ACTION A_Home:
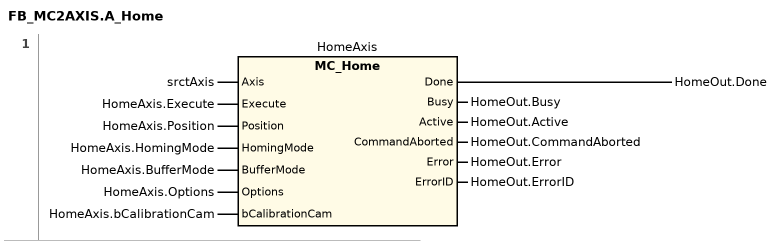
// NETWORK 1
HomeAxis(
    Axis := srctAxis,
    Execute := HomeAxis.Execute,
    Position := HomeAxis.Position,
    HomingMode := HomeAxis.HomingMode,
    BufferMode := HomeAxis.BufferMode,
    Options := HomeAxis.Options,
    bCalibrationCam := HomeAxis.bCalibrationCam,
    Busy => HomeOut.Busy,
    Active => HomeOut.Active,
    CommandAborted => HomeOut.CommandAborted,
    Error => HomeOut.Error,
    ErrorID => HomeOut.ErrorID); // MC_Home
HomeOut.Done := HomeAxis.Done;
END_ACTION

ACTION A_Jog:
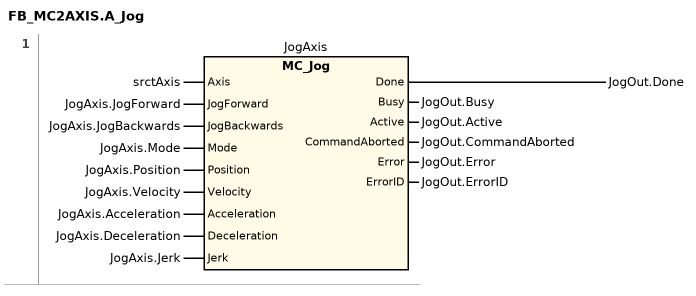
// NETWORK 1
JogAxis(
    Axis := srctAxis,
    JogForward := JogAxis.JogForward,
    JogBackwards := JogAxis.JogBackwards,
    Mode := JogAxis.Mode,
    Position := JogAxis.Position,
    Velocity := JogAxis.Velocity,
    Acceleration := JogAxis.Acceleration,
    Deceleration := JogAxis.Deceleration,
    Jerk := JogAxis.Jerk,
    Busy => JogOut.Busy,
    Active => JogOut.Active,
    CommandAborted => JogOut.CommandAborted,
    Error => JogOut.Error,
    ErrorID => JogOut.ErrorID); // MC_Jog
JogOut.Done := JogAxis.Done;
END_ACTION

ACTION A_MovAbs:
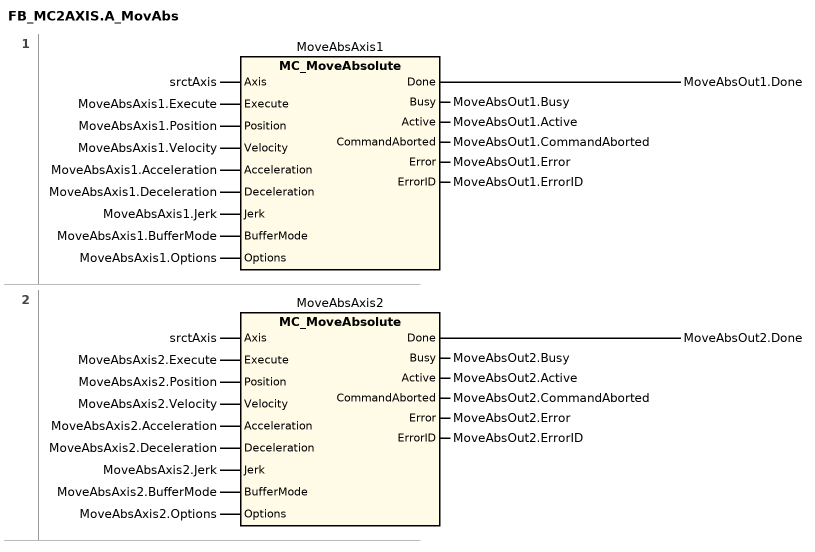
// NETWORK 1
MoveAbsAxis1(
    Axis := srctAxis,
    Execute := MoveAbsAxis1.Execute,
    Position := MoveAbsAxis1.Position,
    Velocity := MoveAbsAxis1.Velocity,
    Acceleration := MoveAbsAxis1.Acceleration,
    Deceleration := MoveAbsAxis1.Deceleration,
    Jerk := MoveAbsAxis1.Jerk,
    BufferMode := MoveAbsAxis1.BufferMode,
    Options := MoveAbsAxis1.Options,
    Busy => MoveAbsOut1.Busy,
    Active => MoveAbsOut1.Active,
    CommandAborted => MoveAbsOut1.CommandAborted,
    Error => MoveAbsOut1.Error,
    ErrorID => MoveAbsOut1.ErrorID); // MC_MoveAbsolute
MoveAbsOut1.Done := MoveAbsAxis1.Done;

// NETWORK 2
MoveAbsAxis2(
    Axis := srctAxis,
    Execute := MoveAbsAxis2.Execute,
    Position := MoveAbsAxis2.Position,
    Velocity := MoveAbsAxis2.Velocity,
    Acceleration := MoveAbsAxis2.Acceleration,
    Deceleration := MoveAbsAxis2.Deceleration,
    Jerk := MoveAbsAxis2.Jerk,
    BufferMode := MoveAbsAxis2.BufferMode,
    Options := MoveAbsAxis2.Options,
    Busy => MoveAbsOut2.Busy,
    Active => MoveAbsOut2.Active,
    CommandAborted => MoveAbsOut2.CommandAborted,
    Error => MoveAbsOut2.Error,
    ErrorID => MoveAbsOut2.ErrorID); // MC_MoveAbsolute
MoveAbsOut2.Done := MoveAbsAxis2.Done;
END_ACTION

ACTION A_MovAdd:
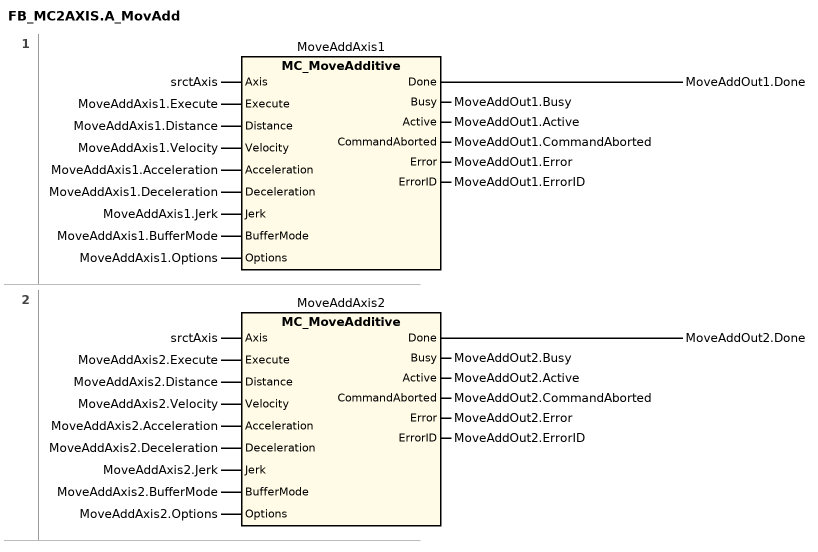
// NETWORK 1
MoveAddAxis1(
    Axis := srctAxis,
    Execute := MoveAddAxis1.Execute,
    Distance := MoveAddAxis1.Distance,
    Velocity := MoveAddAxis1.Velocity,
    Acceleration := MoveAddAxis1.Acceleration,
    Deceleration := MoveAddAxis1.Deceleration,
    Jerk := MoveAddAxis1.Jerk,
    BufferMode := MoveAddAxis1.BufferMode,
    Options := MoveAddAxis1.Options,
    Busy => MoveAddOut1.Busy,
    Active => MoveAddOut1.Active,
    CommandAborted => MoveAddOut1.CommandAborted,
    Error => MoveAddOut1.Error,
    ErrorID => MoveAddOut1.ErrorID); // MC_MoveAdditive
MoveAddOut1.Done := MoveAddAxis1.Done;

// NETWORK 2
MoveAddAxis2(
    Axis := srctAxis,
    Execute := MoveAddAxis2.Execute,
    Distance := MoveAddAxis2.Distance,
    Velocity := MoveAddAxis2.Velocity,
    Acceleration := MoveAddAxis2.Acceleration,
    Deceleration := MoveAddAxis2.Deceleration,
    Jerk := MoveAddAxis2.Jerk,
    BufferMode := MoveAddAxis2.BufferMode,
    Options := MoveAddAxis2.Options,
    Busy => MoveAddOut2.Busy,
    Active => MoveAddOut2.Active,
    CommandAborted => MoveAddOut2.CommandAborted,
    Error => MoveAddOut2.Error,
    ErrorID => MoveAddOut2.ErrorID); // MC_MoveAdditive
MoveAddOut2.Done := MoveAddAxis2.Done;
END_ACTION

ACTION A_MovMod:
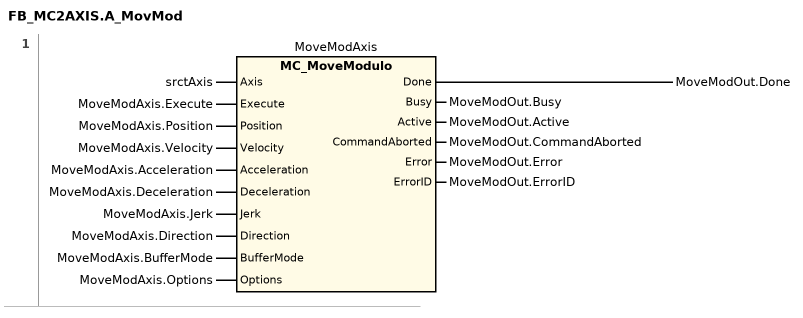
// NETWORK 1
MoveModAxis(
    Axis := srctAxis,
    Execute := MoveModAxis.Execute,
    Position := MoveModAxis.Position,
    Velocity := MoveModAxis.Velocity,
    Acceleration := MoveModAxis.Acceleration,
    Deceleration := MoveModAxis.Deceleration,
    Jerk := MoveModAxis.Jerk,
    Direction := MoveModAxis.Direction,
    BufferMode := MoveModAxis.BufferMode,
    Options := MoveModAxis.Options,
    Busy => MoveModOut.Busy,
    Active => MoveModOut.Active,
    CommandAborted => MoveModOut.CommandAborted,
    Error => MoveModOut.Error,
    ErrorID => MoveModOut.ErrorID); // MC_MoveModulo
MoveModOut.Done := MoveModAxis.Done;
END_ACTION

ACTION A_MovRel:
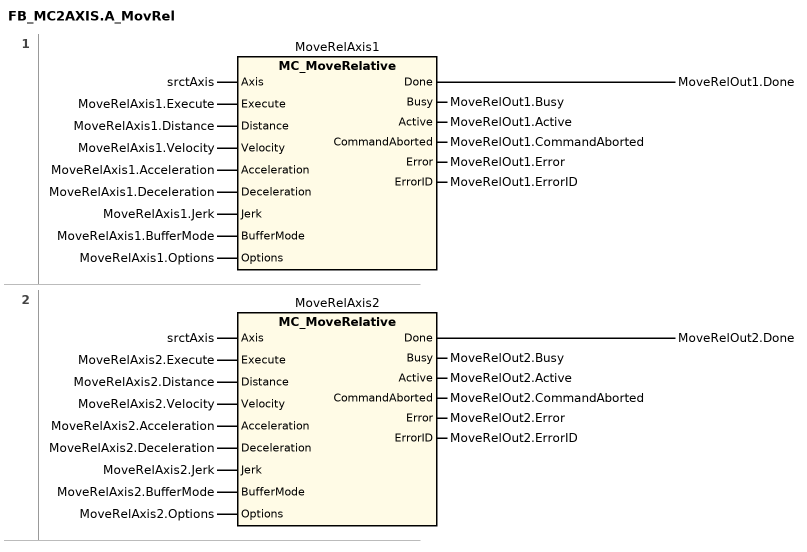
// NETWORK 1
MoveRelAxis1(
    Axis := srctAxis,
    Execute := MoveRelAxis1.Execute,
    Distance := MoveRelAxis1.Distance,
    Velocity := MoveRelAxis1.Velocity,
    Acceleration := MoveRelAxis1.Acceleration,
    Deceleration := MoveRelAxis1.Deceleration,
    Jerk := MoveRelAxis1.Jerk,
    BufferMode := MoveRelAxis1.BufferMode,
    Options := MoveRelAxis1.Options,
    Busy => MoveRelOut1.Busy,
    Active => MoveRelOut1.Active,
    CommandAborted => MoveRelOut1.CommandAborted,
    Error => MoveRelOut1.Error,
    ErrorID => MoveRelOut1.ErrorID); // MC_MoveRelative
MoveRelOut1.Done := MoveRelAxis1.Done;

// NETWORK 2
MoveRelAxis2(
    Axis := srctAxis,
    Execute := MoveRelAxis2.Execute,
    Distance := MoveRelAxis2.Distance,
    Velocity := MoveRelAxis2.Velocity,
    Acceleration := MoveRelAxis2.Acceleration,
    Deceleration := MoveRelAxis2.Deceleration,
    Jerk := MoveRelAxis2.Jerk,
    BufferMode := MoveRelAxis2.BufferMode,
    Options := MoveRelAxis2.Options,
    Busy => MoveRelOut2.Busy,
    Active => MoveRelOut2.Active,
    CommandAborted => MoveRelOut2.CommandAborted,
    Error => MoveRelOut2.Error,
    ErrorID => MoveRelOut2.ErrorID); // MC_MoveRelative
MoveRelOut2.Done := MoveRelAxis2.Done;
END_ACTION

ACTION A_MovVel:
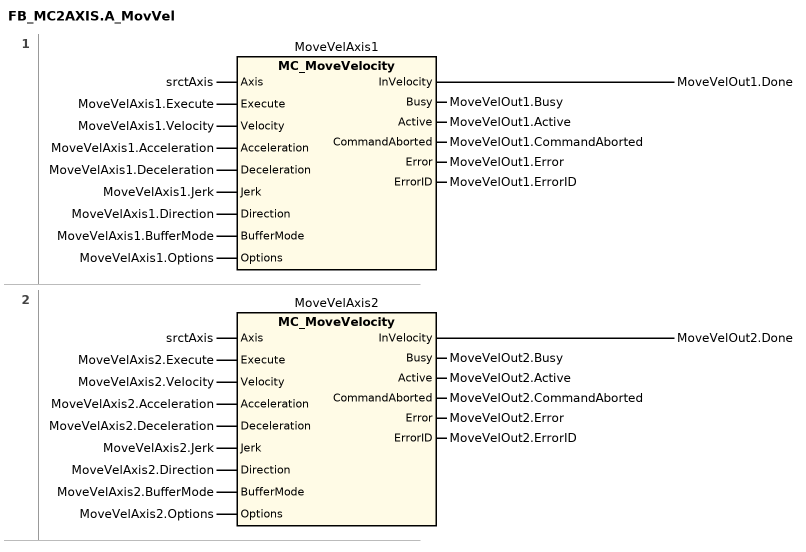
// NETWORK 1
MoveVelAxis1(
    Axis := srctAxis,
    Execute := MoveVelAxis1.Execute,
    Velocity := MoveVelAxis1.Velocity,
    Acceleration := MoveVelAxis1.Acceleration,
    Deceleration := MoveVelAxis1.Deceleration,
    Jerk := MoveVelAxis1.Jerk,
    Direction := MoveVelAxis1.Direction,
    BufferMode := MoveVelAxis1.BufferMode,
    Options := MoveVelAxis1.Options,
    Busy => MoveVelOut1.Busy,
    Active => MoveVelOut1.Active,
    CommandAborted => MoveVelOut1.CommandAborted,
    Error => MoveVelOut1.Error,
    ErrorID => MoveVelOut1.ErrorID); // MC_MoveVelocity
MoveVelOut1.Done := MoveVelAxis1.InVelocity;

// NETWORK 2
MoveVelAxis2(
    Axis := srctAxis,
    Execute := MoveVelAxis2.Execute,
    Velocity := MoveVelAxis2.Velocity,
    Acceleration := MoveVelAxis2.Acceleration,
    Deceleration := MoveVelAxis2.Deceleration,
    Jerk := MoveVelAxis2.Jerk,
    Direction := MoveVelAxis2.Direction,
    BufferMode := MoveVelAxis2.BufferMode,
    Options := MoveVelAxis2.Options,
    Busy => MoveVelOut2.Busy,
    Active => MoveVelOut2.Active,
    CommandAborted => MoveVelOut2.CommandAborted,
    Error => MoveVelOut2.Error,
    ErrorID => MoveVelOut2.ErrorID); // MC_MoveVelocity
MoveVelOut2.Done := MoveVelAxis2.InVelocity;
END_ACTION

ACTION A_Power:

(* read in parameters from the AX5000 via SoE, Reset via SoE *)
fbPowerAxis(
	Enable			:= bEnableAxis,
	Enable_Positive	:= bEnablePos,
	Enable_Negative	:= bEnableNeg,
	Override		:= fOverride,
	Axis			:= srctAxis,
	);

PowerAxisOut.Done := fbPowerAxis.Status;
PowerAxisOut.Busy := fbPowerAxis.Busy;
PowerAxisOut.Active := fbPowerAxis.Active;
PowerAxisOut.Error := fbPowerAxis.Error;
PowerAxisOut.ErrorID := fbPowerAxis.ErrorID;
END_ACTION

ACTION A_ResMovExecute:
HomeAxis.Execute := FALSE;
MoveAbsAxis1.Execute := FALSE;
MoveAbsAxis2.Execute := FALSE;
MoveRelAxis1.Execute := FALSE;
MoveRelAxis2.Execute := FALSE;
MoveAddAxis1.Execute :=FALSE;
MoveAddAxis2.Execute :=FALSE;
MoveVelAxis1.Execute := FALSE;
MoveVelAxis2.Execute := FALSE;
MoveModAxis.Execute := FALSE;
JogAxis.JogBackwards := FALSE;
JogAxis.JogForward := FALSE;
bJogBackwards := FALSE;
bJogForward := FALSE;
END_ACTION

ACTION A_SetPosition:
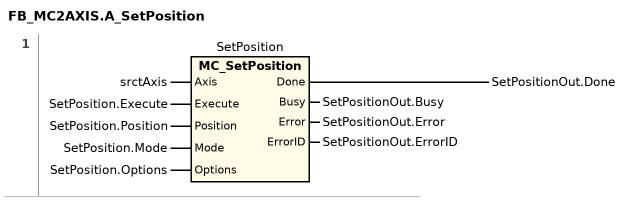
// NETWORK 1
SetPosition(
    Axis := srctAxis,
    Execute := SetPosition.Execute,
    Position := SetPosition.Position,
    Mode := SetPosition.Mode,
    Options := SetPosition.Options,
    Busy => SetPositionOut.Busy,
    Error => SetPositionOut.Error,
    ErrorID => SetPositionOut.ErrorID); // MC_SetPosition
SetPositionOut.Done := SetPosition.Done;
END_ACTION

ACTION A_Stop:
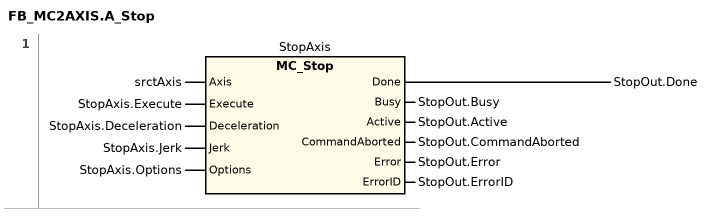
// NETWORK 1
StopAxis(
    Axis := srctAxis,
    Execute := StopAxis.Execute,
    Deceleration := StopAxis.Deceleration,
    Jerk := StopAxis.Jerk,
    Options := StopAxis.Options,
    Busy => StopOut.Busy,
    Active => StopOut.Active,
    CommandAborted => StopOut.CommandAborted,
    Error => StopOut.Error,
    ErrorID => StopOut.ErrorID); // MC_Stop
StopOut.Done := StopAxis.Done;
END_ACTION

ACTION A_Tourque:
(* Tourque and floating axis *)

FromMc2.fActMoment := IiCurrentTourque / 10;

QiTourqueMax := ABS(REAL_TO_INT(fMaxMom * 10));

IF NOT bError AND NOT FromMc2.bError AND srctAxis.Status.Operational AND FloatingCmd.bFloatingOn THEN
	(*	only floating without movement	*)
	IF NOT FloatingCmd.bPush THEN
		fbFloatingAbsAxis1(Execute := FALSE , Axis:=srctAxis);
		fbFloatingAbsAxis2(Execute := FALSE , Axis:=srctAxis);
		fbResetAxisFloating(Execute := (enState = Mc2AxisStateIdle)   , Axis := srctAxis);	(*	AND NOT srctAxis.Status.HasJob	*)
		tonResetFloating(IN := fbResetAxisFloating.Done , PT := T#30ms);
		IF tonResetFloating.Q THEN
			tonResetFloating(IN := FALSE);
			fbResetAxisFloating(Execute := FALSE, Axis := srctAxis);
		END_IF

	(*	floating with negative movement (push)	*)
	ELSIF FloatingCmd.bPush THEN
		fbFloatingMoveTrig(IN := (enState = Mc2AxisStateIdle) , PT := T#200ms);
		IF fbFloatingMoveTrig.Qr THEN
			fbFloatingMoveTrig(IN := FALSE);
			(* FB1 bevorzugen *)
			(* Busy ist high, wenn ein Befehl ansteht; Active ist high, wenn der Mov-Befehl ausgeführt wird *)
			IF NOT fbFloatingAbsAxis1.Busy THEN
				fbFloatingAbsAxis1.Position := srctAxis.NcToPlc.ActPos + FloatingCmd.fPushPos;
				fbFloatingAbsAxis1.Velocity := FloatingCmd.fPushVel;
				fbFloatingAbsAxis1(Execute := TRUE , Axis:=srctAxis);
				fbFloatingAbsAxis2(Execute := FALSE , Axis:=srctAxis);
			(* wenn FB1 aktiv -> neues Kommando mit FB2 überlagern *)
			ELSIF NOT fbFloatingAbsAxis2.Busy THEN
				fbFloatingAbsAxis2.Position := srctAxis.NcToPlc.ActPos + FloatingCmd.fPushPos;
				fbFloatingAbsAxis2.Velocity := FloatingCmd.fPushVel;
				fbFloatingAbsAxis2(Execute := TRUE , Axis:=srctAxis);
				fbFloatingAbsAxis1(Execute := FALSE , Axis:=srctAxis);
			END_IF;
			IF fbFloatingAbsAxis1.Done OR fbFloatingAbsAxis1.CommandAborted OR fbFloatingAbsAxis1.Error THEN
				fbFloatingAbsAxis1(Execute := FALSE , Axis:=srctAxis);
			END_IF
			IF fbFloatingAbsAxis2.Done OR fbFloatingAbsAxis2.CommandAborted OR fbFloatingAbsAxis2.Error THEN
				fbFloatingAbsAxis2(Execute := FALSE , Axis:=srctAxis);
			END_IF
		END_IF
	ELSE
		fbFloatingMoveTrig(IN := FALSE);
		fbFloatingAbsAxis1(Execute := FALSE , Axis:=srctAxis);
		fbFloatingAbsAxis2(Execute := FALSE , Axis:=srctAxis);
	END_IF

	bFederOffReset := FALSE;
ELSE
	fbFloatingMoveTrig(IN := FALSE);
	fbFloatingAbsAxis1(Execute := FALSE , Axis:=srctAxis);
	fbFloatingAbsAxis2(Execute := FALSE , Axis:=srctAxis);
	tonResetFloating(IN := FALSE);
	fbResetAxisFloating(Execute := FALSE, Axis := srctAxis);
	IF NOT bFederOffReset THEN
		fbResetAxisFloating(Execute := TRUE, Axis := srctAxis);
	END_IF
	bFederOffReset := TRUE;
END_IF
fbFloatingAbsAxis1(Axis:=srctAxis );
fbFloatingAbsAxis2(Axis:=srctAxis );
END_ACTION

END_FUNCTION_BLOCK

// Utilities/FB_TON_RMTH
///
///	Dieser Baustein verzögert ein Signal und gibt positive und negative Flanke dieses Signals aus
///	von Roland Ertl / www.rmth.at / 2009
FUNCTION_BLOCK FB_TON_RMTH
VAR_INPUT
	///	Signal	
	IN: BOOL;
	///	Verzögerungszeit	
	PT: TIME := TIME#100ms;
END_VAR
VAR_OUTPUT
	///	Verzögertes Signal	
	Q: BOOL;
	///	Flanken -> nur für 1 Zyklus aktiv	
	Qr: BOOL;
	///	Flanken -> nur für 1 Zyklus aktiv	
	Qf: BOOL;
END_VAR
VAR
	ton_On: TON;
	rtrig_Pos: R_TRIG;
	ftrig_Neg: F_TRIG;
END_VAR

ton_On(IN:= IN , PT:= PT , Q=> Q , ET=> );
rtrig_Pos(CLK:= ton_On.Q , Q=> Qr );
ftrig_Neg(CLK:= ton_On.Q , Q=> Qf);

END_FUNCTION_BLOCK

// Utilities/Balluff/F_GetBalluffWegValue
FUNCTION F_GetBalluffWegValue : REAL
VAR_INPUT
	/// Eingangsdaten von Wegaufnehmer
	arrBytesWeg		:ARRAY[0..3] OF BYTE;
END_VAR
VAR
	nWegTemp		:DWORD;
END_VAR

(*
	Funktion zum mappen der Speicherdaten eines Balluff Wegaufnehmers
	von www.rmth.at/ Roland Ertl / 2015
	Aufloesung 1/1000
	
**********************************************************************)

nWegTemp.0 := arrBytesWeg[3].0;
nWegTemp.1 := arrBytesWeg[3].1;
nWegTemp.2 := arrBytesWeg[3].2;
nWegTemp.3 := arrBytesWeg[3].3;
nWegTemp.4 := arrBytesWeg[3].4;
nWegTemp.5 := arrBytesWeg[3].5;
nWegTemp.6 := arrBytesWeg[3].6;
nWegTemp.7 := arrBytesWeg[3].7;

nWegTemp.8 := arrBytesWeg[2].0;
nWegTemp.9 := arrBytesWeg[2].1;
nWegTemp.10 := arrBytesWeg[2].2;
nWegTemp.11 := arrBytesWeg[2].3;
nWegTemp.12 := arrBytesWeg[2].4;
nWegTemp.13 := arrBytesWeg[2].5;
nWegTemp.14 := arrBytesWeg[2].6;
nWegTemp.15 := arrBytesWeg[2].7;


nWegTemp.16 := arrBytesWeg[1].0;
nWegTemp.17 := arrBytesWeg[1].1;
nWegTemp.18 := arrBytesWeg[1].2;
nWegTemp.19 := arrBytesWeg[1].3;
nWegTemp.20 := arrBytesWeg[1].4;
nWegTemp.21 := arrBytesWeg[1].5;
nWegTemp.22 := arrBytesWeg[1].6;
nWegTemp.23 := arrBytesWeg[1].7;

nWegTemp.24 := arrBytesWeg[0].0;
nWegTemp.25 := arrBytesWeg[0].1;
nWegTemp.26 := arrBytesWeg[0].2;
nWegTemp.27 := arrBytesWeg[0].3;
nWegTemp.28 := arrBytesWeg[0].4;
nWegTemp.29 := arrBytesWeg[0].5;
nWegTemp.30 := arrBytesWeg[0].6;
nWegTemp.31 := arrBytesWeg[0].7;


F_GetBalluffWegValue := DWORD_TO_REAL(nWegTemp) / 1000;

END_FUNCTION

// Utilities/Log/Base/FB_LoggingProviderBase
FUNCTION_BLOCK FB_LoggingProviderBase IMPLEMENTS ITFLoggingProvider

/// Add log method
{attribute '' := ''}
{attribute 'object_name' := 'AddLog'}
METHOD AddLog : BOOL
VAR_INPUT
	/// log message 
	{attribute '' := ''}
	sText: Tc2_System.T_MaxString;
	/// log source
	{attribute '' := ''}
	sSource: STRING;
	///	level: eLogLevelNone, eLogLevelError, eLogLevelWarning, eLogLevelInformation	
	{attribute '' := ''}
	eLevel: E_LogLevel;
END_VAR
VAR
	idx: INT;
END_VAR
///
/// Funktionen zum Hinzufuegen einer Log-Nachricht
/// Rueckgabe: TRUE, bei Erfolg, anderenfalls FALSE
/// 17.05.2010		www.rmth.at
///

idx := iLogArraySize;
REPEAT
	arLoggs[idx] := arLoggs[idx - 1];
    idx:= idx - 1;
UNTIL
    	idx = 0
END_REPEAT

arLoggs[0].sText:= sText;
arLoggs[0].sSource:= sSource;
arLoggs[0].bSaveRequest := TRUE;
arLoggs[0].bSaved  := FALSE;
arLoggs[0].eLevel := eLevel;
arLoggs[0].sTime := sTimeString;

//	Return Result
AddLog := TRUE;
END_METHOD

{attribute 'object_name' := 'Run'}
METHOD Run
END_METHOD

END_FUNCTION_BLOCK

// Utilities/Log/Interface/ITFLoggingProvider
INTERFACE ITFLoggingProvider

/// Add log method
{attribute 'object_name' := 'AddLog'}
METHOD AddLog : BOOL
VAR_INPUT
	/// log message 
	sText: T_MaxString;
	/// log source
	sSource: STRING;
	///	level: eLogLevelNone, eLogLevelError, eLogLevelWarning, eLogLevelInformation	
	eLevel: E_LogLevel;
END_VAR
END_METHOD

{attribute 'object_name' := 'Run'}
METHOD Run
END_METHOD

END_INTERFACE

// Utilities/Log/FB_DebugLoggingProvider
///Funktionblock zum Loggen
FUNCTION_BLOCK FB_DebugLoggingProvider EXTENDS FB_LoggingProviderBase
VAR_IN_OUT
	stLogConfig: ST_LoggingConfig;
END_VAR

///
/// Funktionblock zum Loggen - nur in array
/// 17.05.2010 www.rmth.at
///

END_FUNCTION_BLOCK

// Utilities/Log/FB_EventLoggingProvider
///Funktionblock zum Loggen
FUNCTION_BLOCK FB_EventLoggingProvider EXTENDS FB_LoggingProviderBase
VAR_IN_OUT
	stLogConfig: ST_LoggingConfig;
END_VAR
VAR
	///	logg Message	
	bLoggMessage: BOOL;
	///	input structure		
	strctLogging: ST_Log;
	toiLogging: TON;
	timeLogging: TIME := TIME#2s0ms;
	iLogging: INT;
	ii: INT;
	iSave: INT;
	stEmpty: ST_Log;
	///	MESSAGE ON				
	rtrig_IN: R_TRIG;
	///	message type				
	msgCtrlMask: DWORD;
	///	logging text					
	sText: T_MaxString;
END_VAR

///
/// Funktionblock zum Loggen - windows event log
/// 17.05.2010 www.rmth.at
///

ACTION EventLog:

(*	log trigger	*)
rtrig_IN(clk:= bLoggMessage);

(*	no Log from Configuration	*)
IF stLogConfig.eLogLevel = eLogLevelNone THEN
	bLoggMessage := FALSE;
	RETURN;
END_IF

// switch level
CASE stLogConfig.eLogLevel OF
	eLogLevelInformation:	(*	all eKinds	*)
		IF strctLogging.eLevel = eLogLevelNone THEN
			bLoggMessage := FALSE;
			RETURN;
		END_IF
		
	eLogLevelWarning: 		(*	only Error and Warning	*)
		IF strctLogging.eLevel = eLogLevelNone OR strctLogging.eLevel = eLogLevelInformation THEN
			bLoggMessage := FALSE;
			RETURN;
		END_IF
		
	eLogLevelError: 	(*	only Error	*)
		IF strctLogging.eLevel = eLogLevelNone OR strctLogging.eLevel = eLogLevelInformation OR strctLogging.eLevel = eLogLevelWarning THEN
			bLoggMessage := FALSE;
			RETURN;
		END_IF
		
	ELSE (*	default = none		*)
		bLoggMessage := FALSE;
		RETURN;
		
END_CASE

(*	Event Logg	*)
CASE strctLogging.eLevel OF
	eLogLevelError:	
		msgCtrlMask := 16#14 ; 	(*	Error		*)
	eLogLevelWarning:	
		msgCtrlMask := 16#12;  	(*	Warning		*)
	eLogLevelInformation:
		msgCtrlMask := 16#11;  	(*	Information	*)
ELSE
	msgCtrlMask := 16#11;  	(*	default: Information	*)
END_CASE

IF rtrig_IN.Q THEN
	sText  := strctLogging.sTime;
	sText := CONCAT( sText, ':');
	sText := CONCAT( sText, strctLogging.sSource);
	sText := CONCAT( sText, ':');
	sText := CONCAT( sText, strctLogging.sText);
	ADSLOGSTR(msgCtrlMask,   sText   , '');
END_IF
END_ACTION

ACTION Logger:
///
/// Programm for Logging Messages
/// 11.05.2012	www.rmth.at
///

toiLogging(PT:= timeLogging);

CASE iLogging OF

	0: (*	wait initial Time	*)
		toiLogging.IN := TRUE;
		IF toiLogging.Q THEN
			toiLogging.IN:= FALSE;
			iSave:= 0;
			ii:= 500;
			iLogging := iLogging + 1;
		END_IF

	1: (*	iSave all messages in array list	*)
		CASE iSave OF
			0: 	IF arLoggs[ii].bSaveRequest THEN
					IF  NOT arLoggs[ii].bSaved THEN
						iSave := 10;
					ELSE
						iSave := 100;
					END_IF
				ELSE
					iSave := 100;
				END_IF
	
			10: 	(*	iSave message	*)
				strctLogging := arLoggs[ii];
				bLoggMessage := TRUE;
				iSave:= 11;
	
			11: 	(*	check iSaved	*)
				IF NOT bLoggMessage THEN
					arLoggs[ii].bSaved := TRUE;
					arLoggs[ii].bSaveRequest := FALSE;
					iSave := 100;
				END_IF
	
			100: 	(*	decrement	*)
				ii:= ii - 1;
				iSave := 101;
	
			101:
				IF ii < 0 THEN	(*	all messages checked	*)
					iLogging := iLogging + 1;	(*	next step == clear	*)
				ELSE
					iSave:=0;
				END_IF
		END_CASE

	2: 	(*	delete all iSaved messages	*)
		FOR ii:=0 TO 500 BY 1 DO
			IF arLoggs[ii].bSaved AND NOT arLoggs[ii].bSaveRequest THEN
				arLoggs[ii] := stEmpty;
			END_IF
		END_FOR
		iLogging := 0;

END_CASE
END_ACTION

{attribute 'object_name' := 'Run'}
METHOD Run
Logger();
EventLog();
END_METHOD

END_FUNCTION_BLOCK

// Utilities/Log/FB_FileLoggingProvider
///Funktionblock zum Loggen
FUNCTION_BLOCK FB_FileLoggingProvider EXTENDS FB_LoggingProviderBase
VAR_IN_OUT
	stLogConfig: ST_LoggingConfig;
END_VAR
VAR
	iInit: INT;
	///	logg Message	
	bLoggMessage: BOOL;
	///	input structure		
	strctLogging: ST_Log;
	///	file path example c:\Daten\PLC exist	
	bFilePathExist: BOOL;
	toiLogging: TON;
	timeLogging: TIME := TIME#2s0ms;
	iLogging: INT;
	ii: INT;
	iSave: INT;
	stEmpty: ST_Log;
	///	MESSAGE ON				
	rtrig_IN: R_TRIG;
	///	logging text					
	sText: T_MaxString;
	///	step flow file logging	
	iStepFileLogging: INT;
	hFile: UINT;
	///	full path				
	sPath: STRING;
	///	new full path			
	sPathNew: STRING;
	///	fbs	
	fbFileOpen: FB_FileOpen;
	fbFileWrite: FB_FileWrite;
	bFileWriteBusy: BOOL;
	bFileWriteError: BOOL;
	nFileWriteErrorId: UDINT;
	nFileWriteCount: UDINT;
	fbFileClose: FB_FileClose;
	bFileCloseBusy: BOOL;
	bFileCloseError: BOOL;
	nFileCloseErrorId: UDINT;
	fbEOF: FB_EOF;
	bEOFBusy: BOOL;
	bEOFError: BOOL;
	nEOFErrorId: UDINT;
	///	max file size	
	bIsEOF: BOOL;
	fbFileRename: FB_FileRename;
	bFileRename: BOOL;
	bFileRenameBusy: BOOL;
	bFileRenameError: BOOL;
	nFileRenameErrId: UDINT;
END_VAR

///
/// Funktionblock zum Loggen in Datei
/// 17.05.2010 www.rmth.at
///

{attribute 'object_name' := 'Initialize'}
METHOD PRIVATE Initialize

P_FilePath();

CASE iInit OF
	0:	// path name from configuration
		P_FilePath.sPathName := stLogConfig.sLogPath;
		P_FilePath.bCreateDIR := TRUE;
		iInit := 10;
		
	10:	// wait for folder exists
		IF P_FilePath.bFolderExist THEN
			bFilePathExist := TRUE;
			P_FilePath.bCreateDIR := FALSE;
			iInit := 0;
		END_IF		
END_CASE
END_METHOD

ACTION Logger:
///
/// Programm for Logging Messages
/// 11.05.2012	www.rmth.at
///

toiLogging(PT:= timeLogging);

CASE iLogging OF

	0: (*	wait initial Time	*)
		toiLogging.IN := TRUE;
		IF toiLogging.Q THEN
			toiLogging.IN:= FALSE;
			iSave:= 0;
			ii:= 500;
			iLogging := iLogging + 1;
		END_IF

	1: (*	iSave all messages in array list	*)
		CASE iSave OF
			0: 	IF arLoggs[ii].bSaveRequest THEN
					IF  NOT arLoggs[ii].bSaved THEN
						iSave := 10;
					ELSE
						iSave := 100;
					END_IF
				ELSE
					iSave := 100;
				END_IF
	
			10: 	(*	iSave message	*)
				strctLogging := arLoggs[ii];
				bLoggMessage := TRUE;
				iSave:= 11;
	
			11: 	(*	check iSaved	*)
				IF NOT bLoggMessage THEN
					arLoggs[ii].bSaved := TRUE;
					arLoggs[ii].bSaveRequest := FALSE;
					iSave := 100;
				END_IF
	
			100: 	(*	decrement	*)
				ii:= ii - 1;
				iSave := 101;
	
			101:
				IF ii < 0 THEN	(*	all messages checked	*)
					iLogging := iLogging + 1;	(*	next step == clear	*)
				ELSE
					iSave:=0;
				END_IF
		END_CASE

	2: 	(*	delete all iSaved messages	*)
		FOR ii:=0 TO 500 BY 1 DO
			IF arLoggs[ii].bSaved AND NOT arLoggs[ii].bSaveRequest THEN
				arLoggs[ii] := stEmpty;
			END_IF
		END_FOR
		iLogging := 0;

END_CASE
END_ACTION

{attribute 'object_name' := 'Run'}
METHOD Run
IF NOT bFilePathExist THEN
	Initialize();	
	RETURN;
END_IF

Logger();
WriteFile();
END_METHOD

ACTION WriteFile:

(*	run function logging	*)

(*	trigger	*)
rtrig_IN(clk:= bLoggMessage);

(*	no Log from Configuration	*)
IF stLogConfig.eLogLevel = eLogLevelNone THEN
	bLoggMessage := FALSE;
	RETURN;
END_IF

CASE stLogConfig.eLogLevel OF
	eLogLevelInformation:	(*	all eKinds	*)
		IF strctLogging.eLevel = eLogLevelNone THEN
			bLoggMessage := FALSE;
			RETURN;
		END_IF
	eLogLevelWarning: 		(*	only Error and Warning	*)
		IF strctLogging.eLevel = eLogLevelNone OR strctLogging.eLevel = eLogLevelInformation THEN
			bLoggMessage := FALSE;
			RETURN;
		END_IF
	eLogLevelError: 	(*	only Error	*)
		IF strctLogging.eLevel = eLogLevelNone OR strctLogging.eLevel = eLogLevelInformation OR strctLogging.eLevel = eLogLevelWarning THEN
			bLoggMessage := FALSE;
			RETURN;
		END_IF
	ELSE (*	default = none		*)
		bLoggMessage := FALSE;
		RETURN;
END_CASE

(*	FILE LOG	*)
sPath := '';
sPath := CONCAT(stLogConfig.sLogPath, '\');
sPath := CONCAT(sPath, stLogConfig.sLogName);

sPathNew := '';
sPathNew := CONCAT(stLogConfig.sLogPath, '\');
(*sTimeString:= DELETE(sTimeString,10,10);*)

sPathNew := CONCAT(sPathNew, sTimeString);
sPathNew := CONCAT(sPathNew,'.log');

IF bFilePathExist THEN

	CASE strctLogging.eLevel OF
		eLogLevelError:			(*	Erro		*)
			sText := '$R$N ERR ';
		eLogLevelWarning:		(*	Warning		*)	
			sText := '$R$N WARN ';
		eLogLevelInformation:	(*	info		*)	
			sText := '$R$N INF ';
	ELSE						(*	default		*)				
			sText := '$R$N INF ';
	END_CASE

	sText := CONCAT(sText, strctLogging.sTime);
	sText := CONCAT(sText, ' ');
	sText := CONCAT(sText, strctLogging.sSource);
	sText := CONCAT(sText, ': ');
	sText := CONCAT(sText, strctLogging.sText);

	CASE iStepFileLogging OF

	0: (*	wait for request	*)
		IF rtrig_IN.Q THEN
			hFile := 0; (*	empty File Handle	*)
			fbFileOpen(bExecute:= FALSE);
			iStepFileLogging :=10;
		END_IF

	10: (*	open file	*)
		fbFileOpen(	sNetId:= '',
					sPathName:= sPath ,
					nMode:= FOPEN_MODEAPPEND OR  FOPEN_MODEPLUS,
					ePath:= PATH_GENERIC ,
					bExecute:=TRUE ,
					tTimeout:= t#2s ,
					hFile=> hFile);

		IF NOT fbFileOpen.bBusy THEN
			IF NOT fbFileOpen.bError THEN
				fbFileOpen(bExecute:= FALSE);
				fbFileWrite(bExecute:= FALSE, pWriteBuff := 0, cbWriteLen:=0 );
				fbEOF(bExecute:= FALSE);
				fbFileRename(bExecute:= FALSE);
				iStepFileLogging :=20;
			ELSE
				fbFileOpen(bExecute:= FALSE);
				iStepFileLogging := 0; (*	error	*)
			END_IF
		END_IF

	20: (*	check end of file (max size)	*)
		fbEOF(	hFile:= hFile ,
				bExecute:= TRUE ,
				tTimeout:= t#2s,
				bBusy=> bEOFBusy ,
				bError=> bEOFError ,
				nErrId=> nEOFErrorId ,
				bEOF=> bIsEOF);

		IF NOT fbEOF.bBusy THEN
			IF NOT fbEOF.bError THEN
				fbEOF(bExecute:= FALSE);
				fbFileWrite(bExecute:= FALSE);
				IF NOT bIsEOF THEN
					iStepFileLogging :=30;
				ELSE
					fbFileClose(bExecute:= FALSE);
					iStepFileLogging :=25;
				END_IF
			ELSE
				fbEOF(bExecute:= FALSE);
				iStepFileLogging := 0; (*	error	*)
			END_IF
		END_IF

	25: (*	close file for rename	*)
		fbFileClose(
				sNetId:='' ,
				hFile:=hFile ,
				bExecute:=TRUE ,
				tTimeout:= t#2s,
				bBusy=>bFileCloseBusy ,
				bError=>bFileCloseError ,
				nErrId=>nFileCloseErrorId );

		IF NOT fbFileClose.bBusy THEN
			IF NOT fbFileClose.bError THEN
				fbFileClose(bExecute:= FALSE);
				fbFileRename(bExecute:= FALSE);
				iStepFileLogging := 27;
			ELSE
				fbFileClose(bExecute:= FALSE);
				iStepFileLogging := 0;
			END_IF
		END_IF

	27: (*	Rename full file	*)
		fbFileRename(
				sOldName:= sPath,
				sNewName:=sPathNew ,
				ePath:=PATH_GENERIC ,
				bExecute:= TRUE ,
				tTimeout:= t#2s,
				bBusy=>bFileRenameBusy ,
				bError=>bFileRenameError ,
				nErrId=>nFileRenameErrId );

		IF NOT fbFileRename.bBusy THEN
			IF NOT fbFileRename.bError THEN
				fbFileRename(bExecute:= FALSE);
				iStepFileLogging := 10; (*	new try	*)
			ELSE
				fbFileRename(bExecute:= FALSE);
				iStepFileLogging := 0;
			END_IF
		END_IF

	30: (*	write Data	*)
		fbFileWrite(
				sNetId:='' ,
				hFile:= hFile,
				pWriteBuff:=ADR(sText) ,
				cbWriteLen:= INT_TO_UINT(LEN(sText)),
				bExecute:=TRUE,
				tTimeout:= t#2s ,
				bBusy=>bFileWriteBusy ,
				bError=>bFileWriteError ,
				nErrId=>nFileWriteErrorId ,
				cbWrite=>nFileWriteCount );

		IF NOT fbFileWrite.bBusy THEN
			IF NOT fbFileWrite.bError THEN
				fbFileWrite(bExecute:= FALSE);
				fbFileClose(bExecute:= FALSE);
				iStepFileLogging :=40;
			ELSE
				fbFileWrite(bExecute:= FALSE);
				iStepFileLogging := 0; (*	error	*)
			END_IF
		END_IF

	40: (*	File Close	*)
		fbFileClose(
				sNetId:='' ,
				hFile:=hFile ,
				bExecute:=TRUE ,
				tTimeout:= t#2s,
				bBusy=>bFileCloseBusy ,
				bError=>bFileCloseError ,
				nErrId=>nFileCloseErrorId );

		IF NOT fbFileClose.bBusy THEN
			IF NOT fbFileClose.bError THEN
				fbFileClose(bExecute:= FALSE);
				iStepFileLogging := 0; (*	done	*)
			ELSE
				fbFileClose(bExecute:= FALSE);
				iStepFileLogging := 0; (*	error	*)
			END_IF
		END_IF
	END_CASE
END_IF

(*	clear request for log	*)
IF (iStepFileLogging = 0) THEN
	bLoggMessage := FALSE;
END_IF
END_ACTION

END_FUNCTION_BLOCK

// Utilities/System/P_FilePath
///Programm für die Verzeichnisverwaltung
PROGRAM P_FilePath
VAR_INPUT
	///	path name	
	sPathName: STRING;
	/// 	file name		
	sFileName: STRING;
	///	flag create folder	
	bCreateDIR: BOOL;
	///	flag remove folder	
	bRemoveDIR: BOOL;
END_VAR
VAR_OUTPUT
	///	folder exists flag	
	bFolderExist: BOOL;
END_VAR
VAR
	bBootFolder: BOOL;
	/// 	folders root path 	
	ePath: E_OpenPath;
	///	create DIR	
	fbCreateDir: FB_CreateDir;
	bCreate_Busy: BOOL;
	bCreate_Error: BOOL;
	iCreate_ErrID: UDINT;
	///	delete DIR	
	fbRemoveDir: FB_RemoveDir;
	bRemove_Busy: BOOL;
	bRemove_Error: BOOL;
	iRemove_ErrID: UDINT;
	///	loop		
	iDIR: INT;
END_VAR

///
/// Programm für die Verzeichnisverwaltung
/// 11.05.2012	www.rmth.at
///
(*
	File access program.
	This program is responsible for creating or deleting files.

	Christian Kalser / www.rmth.at / 05.2010
	
	Version:
		0.0.0.1 - Initial Version
*)
(****************************************************************************************)

(*	run program file path	*)
ePath := SEL( bBootFolder, PATH_GENERIC, PATH_BOOTPATH );

CASE iDIR OF

0:
	IF bCreateDIR THEN
		bFolderExist := FALSE;
		bCreateDIR := FALSE;
		fbCreateDir( bExecute := FALSE );
		iDIR := 10;
	ELSIF bRemoveDIR THEN
		bRemoveDIR := FALSE;
		fbRemoveDir( bExecute := FALSE );
		iDIR := 20;
	ELSE
		fbCreateDir( bExecute := FALSE, bBusy=>bCreate_Busy, bError=>bCreate_Error, nErrId=>iCreate_ErrID );
		fbRemoveDir( bExecute := FALSE, bBusy=>bRemove_Busy, bError=>bRemove_Error, nErrId=>iRemove_ErrID );
	END_IF

(*	CREATE DIR		*)
10:
	fbCreateDir(sNetId:= '',
		sPathName:= sPathName,
		ePath:= ePath,
		bExecute:= TRUE,
		tTimeout:= DEFAULT_ADS_TimeOUT,
		bBusy=>bCreate_Busy, bError=>bCreate_Error, nErrId=>iCreate_ErrID );
		iDIR := 12;

12: 	(*	catch error	*)
	fbCreateDir( bExecute := FALSE, bBusy=>bCreate_Busy, bError=>bCreate_Error, nErrId=>iCreate_ErrID );
	IF NOT fbCreateDir.bBusy THEN
		IF NOT fbCreateDir.bError THEN
			bFolderExist := TRUE;
			iDIR := 0;
		ELSE
			CASE iCreate_ErrID OF
				1804: 	(*	folder allready exist	*)
				bFolderExist := TRUE;
				iDIR := 0;
			ELSE
				bFolderExist := FALSE;
				iDIR := 0;
			END_CASE
		END_IF
	END_IF

(*	REMOVE DIR	*)
20:
	fbRemoveDir(sNetId:= '',
		sPathName:= sPathName,
		ePath:= ePath,
		bExecute:= TRUE,
		tTimeout:= DEFAULT_ADS_TimeOUT,
		bBusy=>bRemove_Busy, bError=>bRemove_Error, nErrId=>iRemove_ErrID );
		iDIR := 22;

22: (*	catch error	*)
	fbRemoveDir( bExecute := FALSE, bBusy=>bRemove_Busy, bError=>bRemove_Error, nErrId=>iRemove_ErrID );
	IF NOT fbRemoveDir.bBusy THEN
		IF NOT fbRemoveDir.bError THEN
			bFolderExist := FALSE;
			iDIR := 0;
		ELSE
			CASE iRemove_ErrID OF
				1804:	(*	folder not found	*)
				bFolderExist := FALSE;
				iDIR := 0;
			ELSE
				;
			END_CASE
		END_IF
	END_IF
END_CASE

END_PROGRAM

// Utilities/Math/F_GrayCodeToDecimal
FUNCTION F_GrayCodeToDecimal : BYTE
VAR_INPUT
	nGrayCode: BYTE;
END_VAR
VAR
	ii: INT;
	bB: BOOL;
	bG: BOOL;
END_VAR

// converts the gray code byte to a decimal byte
F_GrayCodeToDecimal:=0;
FOR ii:=7 TO 0 BY -1 DO
	bG:=(nGrayCode AND REAL_TO_BYTE(EXPT(2, ii))) > 0;
	bB:=bB XOR bG;
	F_GrayCodeToDecimal:=F_GrayCodeToDecimal OR SHL(SEL(bB, 2#0, 2#1), ii); 
END_FOR

END_FUNCTION

// Utilities/StringFunctions/StringFunctions/Concat10
FUNCTION Concat10 : T_MaxString
VAR_INPUT
	sExpression1: T_maxString;
	sExpression2: T_maxString;
	sExpression3: T_maxString;
	sExpression4: T_maxString;
	sExpression5: T_maxString;
	sExpression6: T_maxString;
	sExpression7: T_maxString;
	sExpression8: T_maxString;
	sExpression9: T_maxString;
	sExpression10: T_maxString;
END_VAR

Concat10 := CONCAT(sExpression1, sExpression2);
Concat10 := CONCAT(Concat10, sExpression3);
Concat10 := CONCAT(Concat10, sExpression4);
Concat10 := CONCAT(Concat10, sExpression5);
Concat10 := CONCAT(Concat10, sExpression6);
Concat10 := CONCAT(Concat10, sExpression7);
Concat10 := CONCAT(Concat10, sExpression8);
Concat10 := CONCAT(Concat10, sExpression9);
Concat10 := CONCAT(Concat10, sExpression9);
Concat10 := CONCAT(Concat10, sExpression10);

END_FUNCTION

// Utilities/StringFunctions/StringFunctions/Concat2
FUNCTION Concat2 : T_MaxString
VAR_INPUT
	sExpression1: T_maxString;
	sExpression2: T_maxString;
END_VAR

Concat2 := CONCAT(sExpression1, sExpression2);

END_FUNCTION

// Utilities/StringFunctions/StringFunctions/Concat3
FUNCTION Concat3 : T_MaxString
VAR_INPUT
	sExpression1: T_maxString;
	sExpression2: T_maxString;
	sExpression3: T_maxString;
END_VAR

Concat3 := CONCAT(sExpression1, sExpression2);
Concat3 := CONCAT(Concat3, sExpression3);

END_FUNCTION

// Utilities/StringFunctions/StringFunctions/Concat4
FUNCTION Concat4 : T_MaxString
VAR_INPUT
	sExpression1: T_maxString;
	sExpression2: T_maxString;
	sExpression3: T_maxString;
	sExpression4: T_maxString;
END_VAR

Concat4 := CONCAT(sExpression1, sExpression2);
Concat4 := CONCAT(Concat4, sExpression3);
Concat4 := CONCAT(Concat4, sExpression4);

END_FUNCTION

// Utilities/StringFunctions/StringFunctions/Concat5
FUNCTION Concat5 : T_MaxString
VAR_INPUT
	sExpression1: T_maxString;
	sExpression2: T_maxString;
	sExpression3: T_maxString;
	sExpression4: T_maxString;
	sExpression5: T_maxString;
END_VAR

Concat5 := CONCAT(sExpression1, sExpression2);
Concat5 := CONCAT(Concat5, sExpression3);
Concat5 := CONCAT(Concat5, sExpression4);
Concat5 := CONCAT(Concat5, sExpression5);

END_FUNCTION

// Utilities/StringFunctions/StringFunctions/Concat6
FUNCTION Concat6 : T_MaxString
VAR_INPUT
	sExpression1: T_maxString;
	sExpression2: T_maxString;
	sExpression3: T_maxString;
	sExpression4: T_maxString;
	sExpression5: T_maxString;
	sExpression6: T_maxString;
END_VAR

Concat6 := CONCAT(sExpression1, sExpression2);
Concat6 := CONCAT(Concat6, sExpression3);
Concat6 := CONCAT(Concat6, sExpression4);
Concat6 := CONCAT(Concat6, sExpression5);
Concat6 := CONCAT(Concat6, sExpression6);

END_FUNCTION

// Utilities/StringFunctions/StringFunctions/Concat7
FUNCTION Concat7 : T_MaxString
VAR_INPUT
	sExpression1: T_maxString;
	sExpression2: T_maxString;
	sExpression3: T_maxString;
	sExpression4: T_maxString;
	sExpression5: T_maxString;
	sExpression6: T_maxString;
	sExpression7: T_maxString;
END_VAR

Concat7 := CONCAT(sExpression1, sExpression2);
Concat7 := CONCAT(Concat7, sExpression3);
Concat7 := CONCAT(Concat7, sExpression4);
Concat7 := CONCAT(Concat7, sExpression5);
Concat7 := CONCAT(Concat7, sExpression6);
Concat7 := CONCAT(Concat7, sExpression7);

END_FUNCTION

// Utilities/StringFunctions/StringFunctions/Concat8
FUNCTION Concat8 : T_MaxString
VAR_INPUT
	sExpression1: T_maxString;
	sExpression2: T_maxString;
	sExpression3: T_maxString;
	sExpression4: T_maxString;
	sExpression5: T_maxString;
	sExpression6: T_maxString;
	sExpression7: T_maxString;
	sExpression8: T_maxString;
END_VAR

Concat8 := CONCAT(sExpression1, sExpression2);
Concat8 := CONCAT(Concat8, sExpression3);
Concat8 := CONCAT(Concat8, sExpression4);
Concat8 := CONCAT(Concat8, sExpression5);
Concat8 := CONCAT(Concat8, sExpression6);
Concat8 := CONCAT(Concat8, sExpression7);
Concat8 := CONCAT(Concat8, sExpression8);

END_FUNCTION

// Utilities/StringFunctions/StringFunctions/Concat9
FUNCTION Concat9 : T_MaxString
VAR_INPUT
	sExpression1: T_maxString;
	sExpression2: T_maxString;
	sExpression3: T_maxString;
	sExpression4: T_maxString;
	sExpression5: T_maxString;
	sExpression6: T_maxString;
	sExpression7: T_maxString;
	sExpression8: T_maxString;
	sExpression9: T_maxString;
END_VAR

Concat9 := CONCAT(sExpression1, sExpression2);
Concat9 := CONCAT(Concat9, sExpression3);
Concat9 := CONCAT(Concat9, sExpression4);
Concat9 := CONCAT(Concat9, sExpression5);
Concat9 := CONCAT(Concat9, sExpression6);
Concat9 := CONCAT(Concat9, sExpression7);
Concat9 := CONCAT(Concat9, sExpression8);
Concat9 := CONCAT(Concat9, sExpression9);

END_FUNCTION

// Utilities/StringFunctions/StringFunctions/ConcatArray
FUNCTION ConcatArray : T_MaxString
VAR_INPUT
	sArrExpressions: ARRAY[0..15] OF T_maxString;
END_VAR
VAR
	ii: INT;
END_VAR

ConcatArray := '';

FOR ii:=0 TO 15 DO
	ConcatArray := CONCAT(ConcatArray, sArrExpressions[ii]);
END_FOR

END_FUNCTION

// Utilities/StringFunctions/StringFunctions/FB_GetTimeString
FUNCTION_BLOCK FB_GetTimeString
VAR
	fbPulseGetSystemTime: FB_Pulse;
	fbSystemTime: NT_GetTime;
	sTemp: STRING;
	stTimeStruct: TIMESTRUCT;
END_VAR

///
/// Funktion zum Erzeugen eines Zeitstrings
/// 25.04.2006	RE	www.rmth.at
///

sTemp:='';

// read system time
fbPulseGetSystemTime(tPulseTime:=T#100MS);
fbSystemTime(NETID:='', START:=fbPulseGetSystemTime.Q);
fbSystemTime(START:=FALSE);
stTimeStruct:=fbSystemTime.TIMESTR;

IF (stTimeStruct.wYear = 0 AND stTimeStruct.wMonth = 0 AND stTimeStruct.wDay = 0) THEN
	RETURN;
END_IF

(*	date	*)
sTemp:=CONCAT(sTemp , WORD_TO_STRING(stTimeStruct.wYear));

sTemp:=CONCAT(sTemp , '.');
IF stTimeStruct.wMonth < 10 THEN
	sTemp:=CONCAT(sTemp , '0');
END_IF
sTemp:=CONCAT(sTemp , WORD_TO_STRING(stTimeStruct.wMonth));
sTemp:=CONCAT(sTemp , '.');
IF stTimeStruct.wDay < 10 THEN
	sTemp:=CONCAT(sTemp , '0');
END_IF
sTemp:=CONCAT(sTemp , WORD_TO_STRING(stTimeStruct.wDay));

sTemp:=CONCAT(sTemp , '-');

(*	time	*)
IF stTimeStruct.wHour < 10 THEN
	sTemp:=CONCAT(sTemp , '0');
END_IF
sTemp:=CONCAT(sTemp , WORD_TO_STRING(stTimeStruct.wHour));
sTemp:=CONCAT(sTemp , ':');
IF stTimeStruct.wMinute < 10 THEN
	sTemp:=CONCAT(sTemp , '0');
END_IF
sTemp:=CONCAT(sTemp , WORD_TO_STRING(stTimeStruct.wMinute));
sTemp:=CONCAT(sTemp , ':');
IF stTimeStruct.wSecond < 10 THEN
	sTemp:=CONCAT(sTemp , '0');
END_IF
sTemp:=CONCAT(sTemp , WORD_TO_STRING(stTimeStruct.wSecond));
sTemp:=CONCAT(sTemp , ':');
IF stTimeStruct.wMilliseconds < 10 THEN
	sTemp:=CONCAT(sTemp , '00');
ELSIF stTimeStruct.wMilliseconds < 100 THEN
	sTemp:=CONCAT(sTemp , '0');
END_IF
sTemp:=CONCAT(sTemp , WORD_TO_STRING(stTimeStruct.wMilliseconds));

PROPERTY TimeString : STRING
GET
TimeString:=sTemp;
END_GET
END_PROPERTY

END_FUNCTION_BLOCK

// Utilities/FB_Pulse
/// Function block plusegenerator for synchron or asynchron duty cycles
FUNCTION_BLOCK FB_Pulse
VAR_INPUT
	/// pulse time total
	tPulseTime: TIME;
	/// duty cycle factor 0 - 1
	///	default value: 0.5 (50% duty cycle)
	fDutyCycle: REAL := 0.5;
END_VAR
VAR_OUTPUT
	Q: BOOL;
END_VAR
VAR
	tonPulse: TON;
END_VAR

///
/// Programm for pulse generators
/// 10.02.2010	TP www.rmth.at
///

tonPulse(IN := NOT tonPulse.Q, PT:=(tPulseTime));
fDutyCycle:=MIN(fDutyCycle, 1);
IF fDutyCycle <= 0 THEN
	Q:=FALSE;
ELSE
	Q := tonPulse.ET <= REAL_TO_TIME((TIME_TO_REAL(tPulseTime) * fDutyCycle));
END_IF

END_FUNCTION_BLOCK

// Utilities/System/F_GetAdsPort
/// returns the ADS port number used by the current task
FUNCTION F_GetAdsPort : UINT
VAR
	/// FB to get the index of the current task 
	fbTaskIndex: GETCURTASKINDEX;
END_VAR

fbTaskIndex();
F_GetAdsPort := TwinCAT_SystemInfoVarList._TaskInfo[fbTaskIndex.index].AdsPort;

END_FUNCTION

// Utilities/System/F_GetPlcCycleTime
/// returns the PLC cycle time in seconds for the current task
FUNCTION F_GetPlcCycleTime : LREAL
VAR
	/// cycle time in internal units (parts of 100ns)
	nCycleTime: UDINT;
	/// FB to get the index of the current task 
	fbTaskIndex: GETCURTASKINDEX;
END_VAR

fbTaskIndex();
nCycleTime := TwinCAT_SystemInfoVarList._TaskInfo[fbTaskIndex.index].CycleTime;
F_GetPlcCycleTime := nCycleTime * 1.0E-7;   // Cycle Time is given in parts of 100ns

END_FUNCTION

// Utilities/System/F_GetSystemTime64
/// returns the current system time as a 64 bit integer (one unit is equivalent to 100ns)
FUNCTION F_GetSystemTime64 : ULINT
VAR
	/// lower 32 bit of the current time
	nLow: UDINT;
	/// higher 32 bit of the current time value
	nHigh: UDINT;
	/// FB that returns the current time as 2 x 32 bit 
	fbGetTime: GETSYSTEMTIME;
END_VAR

// get the time
fbGetTime( timeLoDW => nLow, timeHiDW => nHigh );

// build a 64 bit integer 
F_GetSystemTime64 := nHigh;
F_GetSystemTime64 := SHL( F_GetSystemTime64, 32 ) OR nLow;

END_FUNCTION

// Utilities/System/P_System
/// Program for reading general system informations
PROGRAM P_System
VAR
	fbPulseGetSystemTime: FB_Pulse;
	fbSystemTime: NT_GetTime;
	fbGetTimeString: FB_GetTimeString;
	/// FB to get the index of the current task
	fbTaskIndex: GETCURTASKINDEX;
	iLoopCount: DINT;
END_VAR

///
/// Program, für allgemeine Systemprozeduren
/// 03.04.2012	TP	www.rmth.at
///

//	read system time
fbPulseGetSystemTime(tPulseTime:=T#100MS);
fbSystemTime(NETID:=sEmpty, START:=fbPulseGetSystemTime.Q);
fbSystemTime(START:=FALSE);

dtNow := SYSTEMTIME_TO_DT(fbSystemTime.TIMESTR);
fbGetTimeString();
sTimeString := fbGetTimeString.TimeString;

//  read system informations
fbTaskIndex();
stPlcSystemInfo.stPlcAppSystemInfo := TwinCAT_SystemInfoVarList._AppInfo;
stPlcSystemInfo.stPlcTaskSystemInfo := TwinCAT_SystemInfoVarList._TaskInfo[fbTaskIndex.index];
stPlcSystemInfo.fCycleTime := stPlcSystemInfo.stPlcTaskSystemInfo.CycleTime * 1.0E-7;			// Cycle Time is given in parts of [100ns] --> to [s]
stPlcSystemInfo.fLastExecTime := stPlcSystemInfo.stPlcTaskSystemInfo.LastExecTime * 1.0E-7;		// Cycle Time is given in parts of [100ns] --> to [s]

//  create default pulses
iLoopCount		:= (iLoopCount + 1) MOD 100;			// loop
stPulse.bImpulse1000ms	:= (iLoopCount MOD 100) = 1;	// 1000ms impulse
stPulse.bImpulse500ms	:= (iLoopCount MOD 50) = 1; 	// 500ms impulse
stPulse.bImpulse300ms	:= (iLoopCount MOD 30) = 1; 	// 300ms impulse
stPulse.bImpulse200ms	:= (iLoopCount MOD 20) = 1; 	// 200ms impulse
stPulse.bImpulse100ms	:= (iLoopCount MOD 10) = 1; 	// 100ms impulse

IF stPulse.bImpulse1000ms THEN
	stPulse.bToggle1000ms := NOT stPulse.bToggle1000ms;
END_IF

IF stPulse.bImpulse500ms THEN
	stPulse.bToggle500ms := NOT stPulse.bToggle500ms;
END_IF

IF stPulse.bImpulse300ms THEN
	stPulse.bToggle300ms := NOT stPulse.bToggle300ms;
END_IF

IF stPulse.bImpulse200ms THEN
	stPulse.bToggle200ms := NOT stPulse.bToggle200ms;
END_IF

IF stPulse.bImpulse100ms THEN
	stPulse.bToggle100ms := NOT stPulse.bToggle100ms;
END_IF

END_PROGRAM

// Utilities/FB_AsyncDrive
FUNCTION_BLOCK FB_AsyncDrive
VAR_INPUT
	/// component active flag
	bActive				:BOOL;
	/// Gibt an ob ein Fehler autom. quitiert werden soll
	bAutoQuittError		:BOOL := TRUE;
	///Objekt Name
	sName				:STRING;
	///Index des Objekts
	diObjectIndex		:DINT;
	/// Sicherheit = Freigabe von Bewegungen
	bSafetyOk			:BOOL;
	/// Hardware OK
	bPowerSupplyOk		:BOOL;
	
	// Hand
	///Ausgewähltes Objekt in der Visu
	diSelectedObjectIndex	:DINT;
	/// Gibt den Handbetrieb frei
	bEnableManual: BOOL;
	// Handbetrieb nach Positiv
	bManual_Pos: BOOL;
	/// Handbetrieb nach Negativ
	bManual_Neg: BOOL;

END_VAR
VAR_OUTPUT
	/// Fehler
	bError				:BOOL;
	/// Fehlertext
	sErrText			:STRING;
	/// 0=Undefiniert
	/// 1=Fehler
	/// 2=Ein
	/// 3=Aus
	iStatus: INT;
	///Darstellung der Controls für das Object 
	///0=Unsichtbar
	///1=Sichtbar Unselektiert
	///2=Sichtbar Selektiert	
	iVisibleState: INT;	
	
	/// Ausgang Positive Richtung
	bOutputDirPos		:BOOL;
	/// Ausgang Negative Richtung
	bOutputDirNeg		:BOOL;
END_VAR
VAR
	bPos, bNeg			:BOOL;
END_VAR

(*
	Einfacher Ansteuerung von Motoren mit Objektorientierten Funktionen
	TwinCAT 3
	2012-2015 / www.rmth.at / RE
	
*************************************************************************)

// nicht aktiv -> alles löschen und Exit
IF NOT bActive THEN
	bError := FALSE ;
	sErrText := '';
	iStatus := 0;/// 0=Undefiniert
	iVisibleState := 0;
	bOutputDirPos := FALSE;
	bOutputDirNeg := FALSE;
	bPos := FALSE;
	bNeg := FALSE;
	RETURN;
END_IF

// Objekt ausgewaehlt
IF (diObjectIndex = diSelectedObjectIndex) THEN
	iVisibleState := 2;	// 2=Sichtbar Selektiert
ELSE
	iVisibleState := 1;	// 1=Sichtbar Unselektiert
END_IF

// Autom. Fehlerreset wenn Fehler nicht mehr ansteht
IF bAutoQuittError THEN
	bError := FALSE;
END_IF

// Sicherheit
IF NOT bSafetyOk THEN
	bOutputDirPos := FALSE;
	bOutputDirNeg := FALSE;
	bPos := FALSE;
	bNeg := FALSE;

// Versorgung NOK 
ELSIF NOT bPowerSupplyOk THEN
	bOutputDirPos := FALSE;
	bOutputDirNeg := FALSE;
	bPos := FALSE;
	bNeg := FALSE;
	bError := TRUE;
	sErrText := CONCAT('Fehler MS ', sName);
	
// OK
ELSE
	// Hand = Automatikbits aus
	IF bEnableManual THEN
		bPos := FALSE;
		bNeg := FALSE;
	END_IF
	
	// wird ueber die Methoden geschalten
	bOutputDirPos := bPos OR (bEnableManual AND bManual_Pos AND (diObjectIndex = diSelectedObjectIndex));
	bOutputDirNeg := bNeg OR (bEnableManual AND bManual_Neg AND (diObjectIndex = diSelectedObjectIndex));
END_IF


// Status in eine Variable zusammenfassen
IF bError THEN
	iStatus := 1; /// 1=Fehler
ELSIF bOutputDirPos OR bOutputDirNeg THEN
	iStatus := 2; /// 2=Ein
ELSIF NOT bOutputDirPos AND NOT bOutputDirNeg THEN
	iStatus := 3; /// 3=Aus
ELSE
	iStatus := 0; /// 0=Undefiniert
END_IF

///	Anforderung Negative Richtung	
{attribute 'object_name' := 'MoveNeg'}
METHOD MoveNeg : BOOL
bPos := FALSE;
bNeg := TRUE;
END_METHOD

///	Anforderung Positive Richtung	
{attribute 'object_name' := 'MovePos'}
METHOD MovePos : BOOL
bPos := TRUE;
bNeg := FALSE;
END_METHOD

METHOD Reset
VAR
END_VAR
bError := FALSE;
END_METHOD

///	Anforderung Stop	
{attribute 'object_name' := 'Stop'}
METHOD Stop : BOOL
bPos := FALSE;
bNeg := FALSE;
END_METHOD

END_FUNCTION_BLOCK

// Utilities/FB_Cylinder
FUNCTION_BLOCK FB_Cylinder
VAR_IN_OUT
	sErrText: STRING;
	bInHome: BOOL;
END_VAR
VAR_INPUT
	///Objekt Name
	s_Name: STRING;
	///	löschen der Ausgänge	
	b_Clear: BOOL;
	///	Anforderung Zylinder in GRST fahren	
	b_Go_HP: BOOL;
	///	Anforderung Zylinder in AST fahren	
	b_Go_WP: BOOL;
	///	Initialisierung zurücksetzen		
	b_ResetInit: BOOL;
	b_EnableManual: BOOL;
	b_Manual_HP: BOOL;
	b_Manual_WP: BOOL;
	b_Sensor_HP: BOOL;
	b_Sensor_WP: BOOL;
	///	Laufzeitüberw. Ein/Aus	
	bSupervision: BOOL;
	///	Laufzeitüberw. zu E0	
	tSupervTime_E0: TIME := TIME#2s0ms;
	///	Laufzeitüberw. zu E1	
	tSupervTime_E1: TIME := TIME#2s0ms;
	///	Aktiviert ob Zylinder beim ersten mal beidseitig mit Druck beaufschlagt werden soll	
	bEnableInit: BOOL := TRUE;
	///	Zus. Freigabe für HP Ausgang schalten	
	bFreigabeHP: BOOL := TRUE;
	///	Zus. Freigabe für WP Ausgang schalten	
	bFreigabeWP: BOOL := TRUE;
END_VAR
VAR_OUTPUT
	b_in_HP: BOOL;
	b_in_WP: BOOL;
	///	GRST angefahren = Grundstellungsfahrt durchgefuehrt	
	b_HP_OK: BOOL;
	b_Init_OK: BOOL;
	b_Valve_HP: BOOL;
	b_Valve_WP: BOOL;
	///	ES Fehler E0	
	bSupervError_E0: BOOL;
	///	ES Fehler E1	
	bSupervError_E1: BOOL;
	///	ES Fehler E0/E1	
	bSupervError_Ex: BOOL;
	bHomeReq: BOOL;
END_VAR
VAR
	pos_AnfGoAST: R_TRIG;
	pos_AnfGoGRST: R_TRIG;
	i_StepInit: INT := 0;
	verz_Init: TON;
	fbTonSuperv_E0: FB_TON_RMTH;
	fbTonSuperv_E1: FB_TON_RMTH;
	posResetInit: R_TRIG;
END_VAR


pos_AnfGoAST(CLK := b_Go_WP);
pos_AnfGoGRST(CLK := b_Go_HP);
IF pos_AnfGoGRST.Q THEN
	b_Go_WP := FALSE ;
END_IF
IF pos_AnfGoAST.Q THEN
	b_Go_HP := FALSE ;
END_IF


(**)
(*	INIT		*)
IF NOT bEnableInit THEN
	b_Init_OK := TRUE;
END_IF

verz_Init(PT := T#0.5s);

(*	reset Init	*)
posResetInit(CLK := b_ResetInit);
IF posResetInit.Q THEN
	b_Go_HP := FALSE;
	b_Go_WP := FALSE;
	b_Init_OK := FALSE;
END_IF


(**)
(*	löschen der Ausgänge	*)
IF b_Clear THEN
	b_Valve_HP := FALSE;
	b_Valve_WP := FALSE;
	b_Go_WP := FALSE ;
	b_Go_HP := FALSE;
	i_StepInit := 0;

ELSIF b_Init_OK AND i_StepInit = 0 THEN

	(*	home position	*)
	IF b_Go_HP OR (b_EnableManual AND b_Manual_HP) THEN
		b_Valve_HP := TRUE;
		b_Valve_WP := FALSE;
		b_Go_WP := FALSE ;
		b_Go_HP := FALSE;
		b_Manual_WP := FALSE;
		IF (b_EnableManual AND b_Manual_HP) THEN	(*	Home req	*)
			bInHome := FALSE;
			bHomeReq := TRUE;
		END_IF

	(*	work position	*)
	ELSIF b_Go_WP OR (b_EnableManual AND b_Manual_WP) THEN
		b_Valve_HP := FALSE;
		b_Valve_WP := TRUE;
		b_Go_WP := FALSE ;
		b_Go_HP := FALSE ;
		b_Manual_HP := FALSE;
		IF (b_EnableManual AND b_Manual_WP) THEN	(*	Home req	*)
			bInHome := FALSE;
			bHomeReq := TRUE;
		END_IF

	END_IF

ELSE

	(*	GRST oder Init	*)
	CASE i_StepInit OF
		0:
			IF b_Go_HP AND NOT b_Init_OK AND bEnableInit THEN
				i_StepInit := 10;
			ELSIF b_Go_HP THEN
				i_StepInit := 20;
			END_IF
		10:
			b_Valve_HP := TRUE;
			b_Valve_WP := TRUE;
			verz_Init.IN := TRUE;
			IF (verz_Init.Q) THEN
				i_StepInit := 20;
			END_IF
	
		(*	GRST	*)
		20:
			b_Valve_HP := TRUE;
			b_Valve_WP := FALSE;
			i_StepInit := 30;
	
		30:
			b_Init_OK := TRUE;
			b_Go_HP := FALSE;
			IF NOT b_Go_HP THEN
				i_StepInit := 0;
			END_IF

	END_CASE

END_IF

IF bInHome THEN
	bHomeReq := FALSE;
END_IF


(**)
(*	Rückmeldung		*)
b_in_HP := b_Sensor_HP AND NOT b_Sensor_WP AND b_Valve_HP;
b_in_WP := b_Sensor_WP AND NOT b_Sensor_HP AND b_Valve_WP ;
b_HP_OK := b_in_HP AND b_Init_OK;

A_Supervision( );

(**)
(*	Sperren	*)
IF b_Valve_HP AND NOT bFreigabeHP THEN
	b_Valve_HP := FALSE;
	bSupervError_Ex := TRUE;
	sErrText := CONCAT(CONCAT('Zyl: ' , s_Name) , ' / Zyl. gesperrt HP');
END_IF
IF b_Valve_WP AND NOT bFreigabeWP THEN
	b_Valve_WP := FALSE;
	bSupervError_Ex := TRUE;
	sErrText := CONCAT(CONCAT('Zyl: ' , s_Name) , ' / Zyl. gesperrt WP');
END_IF

b_Clear := FALSE;

ACTION A_Supervision:

IF NOT bSupervision THEN
	bSupervError_E0 := FALSE;
	bSupervError_E1 := FALSE;
	bSupervError_Ex := FALSE;
	fbTonSuperv_E0(IN := FALSE );
	fbTonSuperv_E1(IN := FALSE );
	RETURN;
END_IF

fbTonSuperv_E0(
	IN := b_Valve_HP AND NOT b_in_HP ,
	PT := tSupervTime_E0);

fbTonSuperv_E1(
	IN := b_Valve_WP AND NOT b_in_WP ,
	PT := tSupervTime_E1);

IF b_Sensor_HP AND b_Sensor_WP THEN
	bSupervError_E0 := FALSE;
	bSupervError_E1 := FALSE;
	bSupervError_Ex := TRUE;
	sErrText := CONCAT(CONCAT('Zyl: ' , s_Name) , ' / Endschalter ERROR');
ELSIF fbTonSuperv_E0.Q THEN
	bSupervError_E0 := TRUE;
	bSupervError_E1 := FALSE;
	bSupervError_Ex := FALSE;
	sErrText := CONCAT(CONCAT('Zyl: ' , s_Name) , ' / E0 (HP) ERROR');
ELSIF fbTonSuperv_E1.Q THEN
	bSupervError_E0 := FALSE;
	bSupervError_E1 := TRUE;
	bSupervError_Ex := FALSE;
	sErrText := CONCAT(CONCAT('Zyl: ' , s_Name) , ' / E1 (WP) ERROR');
ELSE
	bSupervError_E0 := FALSE;
	bSupervError_E1 := FALSE;
	bSupervError_Ex := FALSE;
END_IF
END_ACTION

END_FUNCTION_BLOCK

// Utilities/FB_CylinderEx
FUNCTION_BLOCK FB_CylinderEx
VAR_IN_OUT
	bInHome: BOOL;
END_VAR
VAR_INPUT
	/// component active flag
	bActive: BOOL;
	/// Gibt an ob ein Fehler autom. quitiert werden soll
	bAutoQuittError		:BOOL := TRUE;
	///Objekt Name
	sName				:STRING;
	///Index des Objekts
	diObjectIndex		:DINT;
	///Ventiltyp
	eValveType			:E_ValveType := E_ValveType.eValvetype_5_2_bi;
	/// Sicherheit = Freigabe von Bewegungen
	bSafetyOk			:BOOL;
	/// Druckluftversorgung OK
	bDruckluftOk		:BOOL;
	
	///	Aktiviert ob Zylinder beim ersten mal beidseitig mit Druck beaufschlagt werden soll (2 getrennte Ventile notwendig)	
	bEnableInit			:BOOL := FALSE;

	// Hand
	///Ausgewähltes Objekt in der Visu
	diSelectedObjectIndex	:DINT;
	/// Gibt den Handbetrieb frei
	bEnableManual: BOOL;
	// Handbetrieb nach GRST
	bManual_HP: BOOL;
	/// Handbetrieb nach AST
	bManual_WP: BOOL;
	
	/// Endschalter GRST
	bSensor_HP: BOOL;
	/// Endschalter AST
	bSensor_WP: BOOL;
	
	///	Laufzeitüberw. Ein/Aus	
	bSupervision: BOOL;
	///	Laufzeitüberw. zu GRST
	tSupervTime_HP: TIME := TIME#2S0MS;
	///	Laufzeitüberw. zu AST
	tSupervTime_WP: TIME := TIME#2S0MS;
	
	///	Zus. Freigabe für HP Ausgang schalten	
	bFreigabe_HP: BOOL := TRUE;
	///	Zus. Freigabe für WP Ausgang schalten	
	bFreigabe_WP: BOOL := TRUE;
END_VAR
VAR_OUTPUT	
	/// Summenfehler
	bError		:BOOL;
	/// Fehlerinformation
	sErrText	:STRING;
	/// 0=Undefiniert
	/// 1=Fehler
	/// 2=In GRST (eingefahren)
	/// 3=In AST (ausgefahren) 
	iStatus: INT;	
	///Darstellung der Controls für das Object 
	///0=Unsichtbar
	///1=Sichtbar Unselektiert
	///2=Sichtbar Selektiert	
	iVisibleState: INT;

	bIn_HP: BOOL;
	bIn_WP: BOOL;
	///	GRST angefahren = Grundstellungsfahrt durchgefuehrt	
	bHP_OK: BOOL;
	bInit_OK: BOOL;
	
	bValve_HP: BOOL;
	bValve_WP: BOOL;
	
	///	ES Fehler GRST	
	bSupervError_HP: BOOL;
	///	ES Fehler AST	
	bSupervError_WP: BOOL;
	///	ES Fehler E0/E1	
	bSupervError_HPWP: BOOL;
	
	/// GRST erforderlich
	bHomeReq: BOOL;
	
	/// Aktuelle Positionen mit gelatchten Objektposition gleich
	bLatchedObjPositionOK					:BOOL;
END_VAR
VAR
	///	löschen der Ausgänge	
	bClear: BOOL;
	///	Anforderung Zylinder in GRST fahren	
	bGo_HP: BOOL;
	///	Anforderung Zylinder in AST fahren	
	bGo_WP: BOOL;

	bMan_HP, bMan_WP	:BOOL;
		
	iStepInit: INT := 0;
	tonInit: TON;
	fbTonSuperv_HP: FB_TON_RMTH;
	fbTonSuperv_WP: FB_TON_RMTH;
	
	iStatusLatched			:INT;
END_VAR

(*
	Einfacher Zylinder Baustein mit Objektorientierten Funktionen
	TwinCAT 3
	2012-2015 / www.rmth.at / RE, TP
	
*************************************************************************)

// nicht aktiv -> alles löschen und Exit
IF NOT bActive THEN
	bError := FALSE ;
	sErrText := '';
	iStatus := 0;/// 0=Undefiniert
	iVisibleState := 0;
	bValve_HP := FALSE;
	bValve_WP := FALSE;
	bGo_WP := FALSE ;
	bGo_HP := FALSE;
	iStepInit := 0;
	bSupervError_HP := FALSE;
	bSupervError_WP := FALSE;
	bSupervError_HPWP := FALSE;
	bHomeReq := FALSE;
	bInit_OK := FALSE;
	RETURN;
END_IF

(**)
(*	INIT		*)
IF NOT bEnableInit THEN
	bInit_OK := TRUE;
END_IF

tonInit(PT := T#0.5S);

// Objekt ausgewaehlt
IF (diObjectIndex = diSelectedObjectIndex) THEN
	iVisibleState := 2;	// 2=Sichtbar Selektiert
ELSE
	iVisibleState := 1;	// 1=Sichtbar Unselektiert
END_IF

(* Sicherheit	*)
IF NOT bSafetyOk THEN
	// TODO: je nach Ventiltyp
	bGo_WP := FALSE ;
	bGo_HP := FALSE;
	iStepInit := 0;

(*	löschen der Ausgänge	*)
ELSIF bClear THEN
	bValve_HP := FALSE;
	bValve_WP := FALSE;
	bGo_WP := FALSE ;
	bGo_HP := FALSE;
	iStepInit := 0;

ELSIF NOT bDruckluftOk THEN
	;
	
ELSIF bInit_OK AND iStepInit = 0 THEN

	bMan_HP := (bEnableManual AND bManual_HP AND (diObjectIndex = diSelectedObjectIndex));
	bMan_WP := (bEnableManual AND bManual_WP AND (diObjectIndex = diSelectedObjectIndex));
	(*	home position	*)
	IF bGo_HP OR bMan_HP THEN
		bValve_HP := TRUE;
		bValve_WP := FALSE;
		bGo_WP := FALSE ;
		bGo_HP := FALSE;
		bManual_WP := FALSE;
		IF bMan_HP THEN	(*	Home req da manuell verfahren	*)
			bInHome := FALSE;
			bHomeReq := TRUE;
		END_IF

	(*	work position	*)
	ELSIF bGo_WP OR bMan_WP THEN
		bValve_HP := FALSE;
		bValve_WP := TRUE;
		bGo_WP := FALSE ;
		bGo_HP := FALSE ;
		bManual_HP := FALSE;
		IF bMan_WP THEN	(*	Home req da manuell verfahren	*)
			bInHome := FALSE;
			bHomeReq := TRUE;
		END_IF

	END_IF

ELSE

	(*	GRST oder Init	*)
	CASE iStepInit OF
		0:
			IF bGo_HP AND NOT bInit_OK AND bEnableInit THEN
				iStepInit := 10;
			ELSIF bGo_HP THEN
				iStepInit := 20;
			END_IF
		10:
			bValve_HP := TRUE;
			bValve_WP := TRUE;
			tonInit.IN := TRUE;
			IF (tonInit.Q) THEN
				iStepInit := 20;
			END_IF
	
		(*	GRST	*)
		20:
			bValve_HP := TRUE;
			bValve_WP := FALSE;
			iStepInit := 30;
	
		30:
			bInit_OK := TRUE;
			bGo_HP := FALSE;
			IF NOT bGo_HP THEN
				iStepInit := 0;
			END_IF

	END_CASE

END_IF

IF bInHome THEN
	bHomeReq := FALSE;
END_IF


(**)
(*	Rückmeldung		*)
bIn_HP := bSensor_HP AND NOT bSensor_WP AND bValve_HP;
bIn_WP := bSensor_WP AND NOT bSensor_HP AND bValve_WP ;
bHP_OK := bIn_HP AND bInit_OK;

A_Supervision( );

(**)
(*	Sperren	*)
IF bValve_HP AND NOT bFreigabe_HP THEN
	bValve_HP := FALSE;
	bSupervError_HPWP := TRUE;
	sErrText := CONCAT(CONCAT('Zyl: ' , sName) , ' / Zyl. gesperrt HP');
END_IF
IF bValve_WP AND NOT bFreigabe_WP THEN
	bValve_WP := FALSE;
	bSupervError_HPWP := TRUE;
	sErrText := CONCAT(CONCAT('Zyl: ' , sName) , ' / Zyl. gesperrt WP');
END_IF

// Summenfehler Fehler
bError := bSupervError_HP OR bSupervError_WP OR bSupervError_HPWP;

// Status in eine Variable zusammenfassen
IF bError THEN 
	iStatus := 1; // 1=Fehler
ELSIF (bSensor_HP AND NOT bSensor_WP) THEN
	iStatus := 2; // 2=In GRST (eingefahren)
ELSIF (bSensor_WP AND NOT bSensor_HP) THEN
	iStatus := 3; // 3=In AST (ausgefahren)
ELSE
	iStatus := 0; // 0=Undefiniert
END_IF

bClear := FALSE;

A_CheckLatchState();

ACTION A_CheckLatchState:
// Status vergleichen
// OR (iStatusLatched = 1)
bLatchedObjPositionOK := iStatusLatched = iStatus OR (iStatusLatched = 1); // Status gleich oder gemerkter Status Fehler
END_ACTION

ACTION A_Supervision:

IF NOT bSupervision THEN
	bSupervError_HP := FALSE;
	bSupervError_WP := FALSE;
	bSupervError_HPWP := FALSE;
	fbTonSuperv_HP(IN := FALSE );
	fbTonSuperv_WP(IN := FALSE );
	RETURN;
END_IF

fbTonSuperv_HP(
	IN := bValve_HP AND NOT bIn_HP ,
	PT := tSupervTime_HP);

fbTonSuperv_WP(
	IN := bValve_WP AND NOT bIn_WP ,
	PT := tSupervTime_WP);

// Autom. Fehlerreset wenn Fehler nicht mehr ansteht
IF bAutoQuittError THEN
	bSupervError_HP := FALSE;
	bSupervError_WP := FALSE;
	bSupervError_HPWP := FALSE;
END_IF	
	
IF bSensor_HP AND bSensor_WP THEN
	bSupervError_HP := FALSE;
	bSupervError_WP := FALSE;
	bSupervError_HPWP := TRUE;
	sErrText := CONCAT(CONCAT('Zyl: ' , sName) , ' / Endschalter ERROR');
ELSIF fbTonSuperv_HP.Q THEN
	bSupervError_HP := TRUE;
	bSupervError_WP := FALSE;
	bSupervError_HPWP := FALSE;
	sErrText := CONCAT(CONCAT('Zyl: ' , sName) , ' / E0 (HP) ERROR');
ELSIF fbTonSuperv_WP.Q THEN
	bSupervError_HP := FALSE;
	bSupervError_WP := TRUE;
	bSupervError_HPWP := FALSE;
	sErrText := CONCAT(CONCAT('Zyl: ' , sName) , ' / E1 (WP) ERROR');
END_IF
END_ACTION

///	löschen der Ausgänge
{attribute 'object_name' := 'ClearOuts'}
METHOD ClearOuts : BOOL
bClear := TRUE;
bGo_HP := FALSE;
bGo_WP := FALSE;
bValve_HP := FALSE;
bValve_WP := FALSE;
END_METHOD

///	Anforderung Zylinder in GRST fahren	
{attribute 'object_name' := 'GoHP'}
METHOD GoHP : BOOL
bGo_HP := TRUE;
bGo_WP := FALSE;
END_METHOD

///	Anforderung Zylinder in AST fahren	
{attribute 'object_name' := 'GoWP'}
METHOD GoWP : BOOL
bGo_HP := FALSE;
bGo_WP := TRUE;
END_METHOD

/// Methode um Status des Objekt zu speichern
METHOD LatchObjState : BOOL
iStatusLatched := iStatus;
END_METHOD

METHOD Reset
VAR
END_VAR
bSupervError_HP := FALSE;
bSupervError_WP := FALSE;
bSupervError_HPWP := FALSE;
END_METHOD

///	Initialisierung zurücksetzen		
{attribute 'object_name' := 'ResetInit'}
METHOD ResetInit : BOOL
bGo_HP := FALSE;
bGo_WP := FALSE;
bInit_OK := FALSE;
END_METHOD

END_FUNCTION_BLOCK

// Utilities/FB_RotaryEncoder
FUNCTION_BLOCK FB_RotaryEncoder
VAR_INPUT
	///Wert von Zählklemme
	Ii_EL5101_Count AT %I*: UINT;
	/// [1.57079E-5] = 0.314m / 20000 (=5000 Strich Geber) Skalierungsfaktor für Ergebniswerte "init für TACHO" 
	f_Skalierungsfaktor: REAL := 1.57079E-05;
	///Setzt den löschbaren Zähler zurück
	b_ResetCount: BOOL;
	///Anforderung auf Position setzen
	b_SetPos: BOOL;
	/// Position, auf die mit SetPos gesetzt wird 
	f_PosSet: REAL;
END_VAR
VAR_OUTPUT
	///Berechneter Messwert \ Länge
	f_Messwert: REAL;
	///Ausgabe der Länge in Increments ==> wird nie genullt!
	i_Messwert_Inc: DINT;
	/// Geschwindigkeit 
	f_Vist: REAL;
	/// Geschwindigkeit aus 100ms Zyklus berechnet 
	f_Vist_100: REAL;
	/// Impuls für 1 Cyklus 
	b_NewSpeed: BOOL;
END_VAR
VAR
	///Hilfvariable für Zählervergleich
	i_Count_old: DINT;
	/// für rücksetzbare Länge 
	i_Count_CanReset: DINT;
	/// für ewige Messung intern 
	i_Count_Ever: DINT;
	/// für Ring Messung intern 
	i_Count_RingTeil: DINT;
	/// Länge alt in Incr für Geschwindigkeit \ 1000ms Task
	i_Messwert_Inc_alt: DINT;
	/// Länge alt in Incr für Geschwindigkeit  \  100ms Task
	i_MW_Inc_alt100: DINT;
	iarrCountSubLaengen: ARRAY[0..20] OF DINT;
	aa: INT;
	bInit: BOOL;
END_VAR


(*	TACHO ROLLE \ PRODUKTIONS Länge u. Geschwindigkeit	*)

(*Initialisierung*)
IF (NOT bInit) THEN
	i_Count_old := Ii_EL5101_Count;	(*aktuelle Zählgröße auf Hilfmerker übertragen*)
	i_Count_CanReset := - UINT_TO_INT(Ii_EL5101_Count) + REAL_TO_DINT(f_Messwert / f_Skalierungsfaktor);  (*Messwert konvertieren zu Zähler Type*)
	i_Count_Ever := - UINT_TO_INT(Ii_EL5101_Count);	(*Befüllen counter für ewige interne Messung*)
	bInit := TRUE;
END_IF

(*Overflow von Value der EL5101 65536 --> 0*)
IF (i_Count_old - Ii_EL5101_Count) > 30000 THEN
	i_Count_CanReset := i_Count_CanReset + 65536;	(*Auflösung von 16Bit = 2^16 = 65536*)
	i_Count_Ever := i_Count_Ever + 65536;
	i_Count_RingTeil := i_Count_RingTeil + 65536;
END_IF

(*Underflow von Value der EL5101 0 --> 65536*)
IF (i_Count_old - Ii_EL5101_Count) < - 30000 THEN
	i_Count_CanReset := i_Count_CanReset - 65536;
	i_Count_Ever := i_Count_Ever - 65536;
	i_Count_RingTeil := i_Count_RingTeil - 65536;
END_IF

(*Wert zum Vergleichen speichern*)
i_Count_old := Ii_EL5101_Count;

(*Externe Anforderung Zähler rücksetzen*)
IF (b_ResetCount) THEN
	i_Count_CanReset := - UINT_TO_INT(Ii_EL5101_Count);
	b_ResetCount:= FALSE; (*Anforderung löscht sich selber*)
END_IF

(*Externe Anforderung Zähler auf eine Position setzen*)
IF (b_SetPos) THEN
	i_Count_CanReset := - UINT_TO_INT(Ii_EL5101_Count) + REAL_TO_INT(f_PosSet / f_Skalierungsfaktor);
	b_SetPos := FALSE; (*Anforderung löscht sich selber*)
END_IF


(*BERECHNUNG LÄNGE*)

(*Messwert für die Länge / Produkt*)
f_Messwert:= DINT_TO_REAL(i_Count_CanReset + Ii_EL5101_Count) * f_Skalierungsfaktor;

(*Messwert in Increments / wird nie genullt*)
i_Messwert_Inc :=	i_Count_Ever + Ii_EL5101_Count;

(* BERECHNUNG GESCHWINDIGKEIT*)

IF (stPulse.bImpulse1000ms) THEN
	f_Vist := DINT_TO_REAL(i_Messwert_Inc - i_Messwert_Inc_alt) * 60 * f_Skalierungsfaktor;
	i_Messwert_Inc_alt := i_Messwert_Inc;
END_IF
b_NewSpeed := stPulse.bImpulse1000ms;

IF (stPulse.bImpulse1000ms) THEN
	f_Vist_100 := DINT_TO_REAL(i_Messwert_Inc - i_MW_Inc_alt100) * 600 * f_Skalierungsfaktor;
	i_MW_Inc_alt100 := i_Messwert_Inc;
END_IF

END_FUNCTION_BLOCK

// Utilities/FB_ScaleAnalogInput
FUNCTION_BLOCK FB_ScaleAnalogInput
VAR_INPUT
	/// Analoge Daten von der Klemme
	iAnalogInputValue	:INT;
	/// Maximalwert
	fMaxVal				:REAL := 100;
	/// Maximalwert des analogen Eingangs
	fAnalogInMaxVal		:REAL := 32767;
END_VAR
VAR_OUTPUT
	/// Skalierter Wert
	fValue				:REAL;
END_VAR
VAR
	fFactor: REAL;
END_VAR


(*Berechnung Skalierungsfaktor*)
fFactor := fMaxVal / fAnalogInMaxVal;

(*Ausgabe der Eingangsdaten in [Bar] *)
fValue := fFactor * INT_TO_REAL(iAnalogInputValue);

END_FUNCTION_BLOCK

// Utilities/FB_Sensor
FUNCTION_BLOCK FB_Sensor
VAR_INPUT
	b_Signal: BOOL;
	tt_SignalFilter: TIME := TIME#30ms;
	tt_SignalFilter_Inv: TIME := TIME#500ms;
END_VAR
VAR_OUTPUT
	///	verzögertes Signal	
	Q: BOOL;
	///	negiertes verzögertes Signal	
	Q_Inv: BOOL;
	///	pos. Flanke von Signal		
	Qr: BOOL;
	///	neg. Flanke von Signal		
	Qf: BOOL;
END_VAR
VAR
	verz_Signal: FB_TON_RMTH;
	verz_Signal_Inv: FB_TON_RMTH;
END_VAR


verz_Signal		(IN := b_Signal, PT := tt_SignalFilter);
verz_Signal_Inv	(IN := NOT b_Signal, PT := tt_SignalFilter_Inv);

Q := verz_Signal.Q;
Qr := verz_Signal.Qr;
Qf := verz_Signal.Qf;

Q_Inv := verz_Signal_Inv.Q;

END_FUNCTION_BLOCK
